PROGRAM CoEConfig
VAR
END_VAR

;

END_PROGRAM

(* stored: Version 1.1.0.1, ProductVersion 3.1.4024.9
   POU CoEConfig: Id {ac67faf6-46b9-4ce7-a6dd-13d16b67c657}, SpecialFunc None *)
